FUNCTION_BLOCK FB_MX2
VAR_INPUT
	b_CW   AT%I*  :BOOL;
	b_CCW AT%I*  :BOOL;
	b_Reset AT%I* :BOOL;
	ui_CzestotliwoscI AT %I*: INT;
	w_Status AT%I* :WORD;
	udi_RampaACC_in AT %I*: WORD;
	udi_RampaDCC_in AT %I*: WORD;
END_VAR
	
	
VAR_OUTPUT
	ui_CzestotliwoscO AT %Q*: INT;
	udi_RampaACC_out AT %Q*: WORD;
	udi_RampaDCC_out AT %Q*: WORD;
	b_Rady AT %Q*: BOOL;
	b_Pracuje AT %Q*: BOOL;
	w_ControlW AT%Q* :WORD;
	Blad AT%Q* :BOOL;
END_VAR

VAR
	
	LokRem : BOOL;
	DoPrzodu :BOOL;
	DoTylu:BOOL;
	BladFalownik :BOOL;
	BladFalownikKom :BOOL;
	out1 :WORD;
	out2 :WORD;
	out3 :WORD;
	out4 :WORD;
	out5 :WORD;
	OP_O :TON;
	axal_Fal : BOOL;
	OP_50Hax : TON;
	OP_Hax :TON;
	Fal_s :INT;
	OP_Falownik_OFF :TON;
	Wyl_Fal :BOOL;
	
	
	
	Wylacz: BOOL;
END_VAR

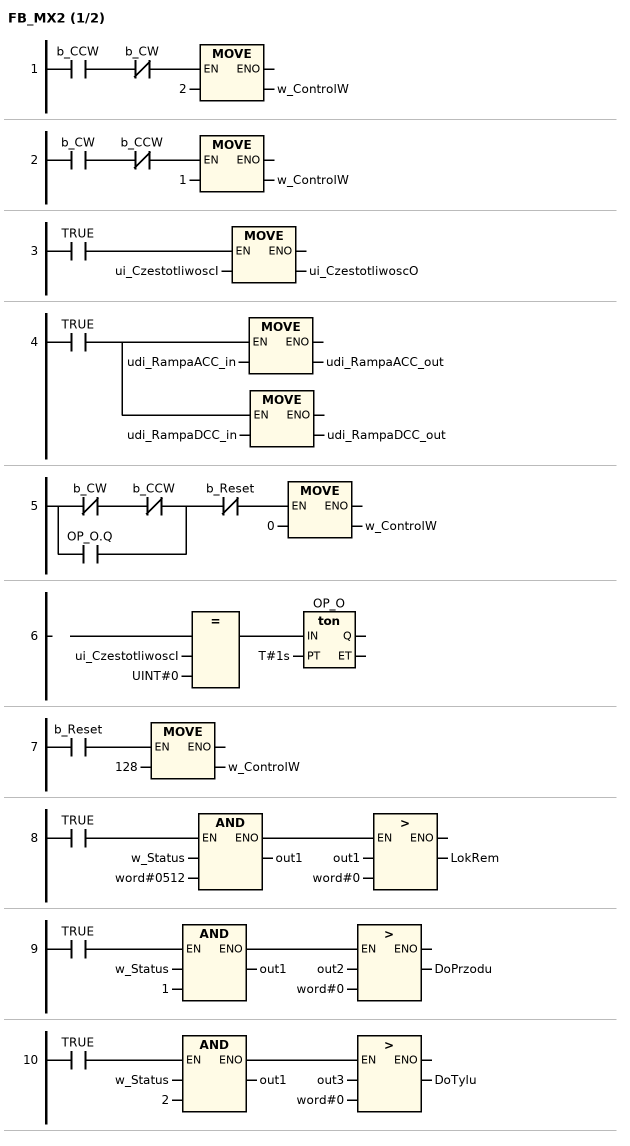
// NETWORK 1
IF b_CCW AND NOT b_CW THEN w_ControlW := 2; END_IF

// NETWORK 2
IF b_CW AND NOT b_CCW THEN w_ControlW := 1; END_IF

// NETWORK 3
ui_CzestotliwoscO := ui_CzestotliwoscI;

// NETWORK 4
udi_RampaACC_out := udi_RampaACC_in;
udi_RampaDCC_out := udi_RampaDCC_in;

// NETWORK 5
IF (NOT b_CW AND NOT b_CCW OR OP_O.Q) AND NOT b_Reset THEN w_ControlW := 0; END_IF

// NETWORK 6
OP_O(IN := ui_CzestotliwoscI = UINT#0, PT := T#1s); // ton

// NETWORK 7
IF b_Reset THEN w_ControlW := 128; END_IF

// NETWORK 8
out1 := w_Status AND word#0512;
LokRem := out1 > word#0;

// NETWORK 9
out1 := w_Status AND 1;
DoPrzodu := out2 > word#0;

// NETWORK 10
out1 := w_Status AND 2;
DoTylu := out3 > word#0;

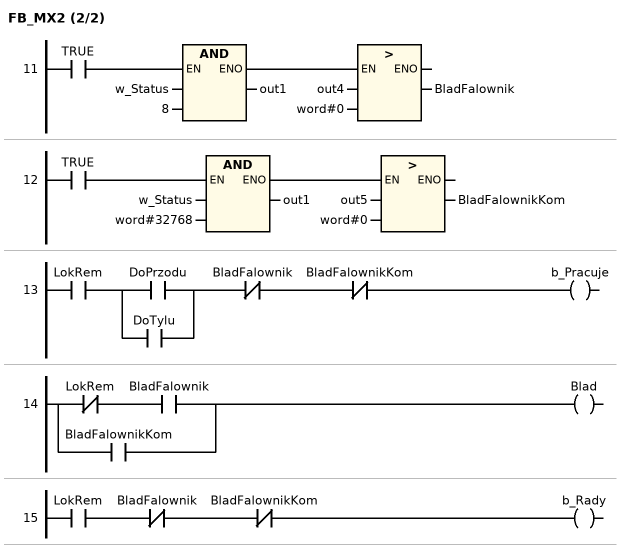
// NETWORK 11
out1 := w_Status AND 8;
BladFalownik := out4 > word#0;

// NETWORK 12
out1 := w_Status AND word#32768;
BladFalownikKom := out5 > word#0;

// NETWORK 13
b_Pracuje := LokRem AND (DoPrzodu OR DoTylu) AND NOT BladFalownik AND NOT BladFalownikKom;

// NETWORK 14
Blad := NOT LokRem AND BladFalownik OR BladFalownikKom;

// NETWORK 15
b_Rady := LokRem AND NOT BladFalownik AND NOT BladFalownikKom;

END_FUNCTION_BLOCK

(* stored: Version 1.1.0.1, ProductVersion 3.1.4022.12
   POU FB_MX2: Id {61d8f789-0d78-4f3e-b403-e55cdc640241}, SpecialFunc None *)
